// Mitsubishi GX Works2 project: BookEX6_5 Shift   PLC: Q06UDV

// global labels: Global
VAR_GLOBAL
  bVar0 AT M5000 : BOOL;
  abArray0 AT M5010 : ARRAY [0..49] OF BOOL;
  sStr0 AT D5000 : STRING[199];
  sStr1 AT D5100 : STRING[199];
  sStr2 AT D5200 : STRING[199];
  sStr3 AT D5300 : STRING[199];
  sStr4 AT D5400 : STRING[199];
  sStr5 AT D5500 : STRING[199];
  sStr6 AT D5600 : STRING[199];
  sStr7 AT D5700 : STRING[199];
  sStr8 AT D5800 : STRING[199];
  sStr9 AT D5900 : STRING[199];
  iVar0 AT D4500 : INT;
  iVar1 AT D4501 : INT;
  iVar2 AT D4502 : INT;
  iVar3 AT D4503 : INT;
  iVar4 AT D4504 : INT;
  iVar5 AT D4505 : INT;
  iVar6 AT D4506 : INT;
  iVar7 AT D4507 : INT;
  iVar8 AT D4508 : INT;
  iVar9 AT D4509 : INT;
  dVar0 AT D4510 : DINT;
  dVar1 AT D4512 : DINT;
  dVar2 AT D4514 : DINT;
  dVar3 AT D4516 : DINT;
  dVar4 AT D4518 : DINT;
  dVar5 AT D4520 : DINT;
  dVar6 AT D4522 : DINT;
  dVar7 AT D4524 : DINT;
  dVar8 AT D4526 : DINT;
  dVar9 AT D4528 : DINT;
  wVar0 AT D4530 : WORD;
  wVar1 AT D4531 : WORD;
  wVar2 AT D4532 : WORD;
  wVar3 AT D4533 : WORD;
  wVar4 AT D4534 : WORD;
  wVar5 AT D4535 : WORD;
  wVar6 AT D4536 : WORD;
  wVar7 AT D4537 : WORD;
  wVar8 AT D4538 : WORD;
  wVar9 AT D4539 : WORD;
  dwVar0 AT D4540 : DWORD;
  dwVar1 AT D4542 : DWORD;
  dwVar2 AT D4544 : DWORD;
  dwVar3 AT D4546 : DWORD;
  dwVar4 AT D4548 : DWORD;
  dwVar5 AT D4550 : DWORD;
  dwVar6 AT D4552 : DWORD;
  dwVar7 AT D4554 : DWORD;
  dwVar8 AT D4556 : DWORD;
  dwVar9 AT D4558 : DWORD;
  fsVar0 AT D4560 : REAL;
  fsVar1 AT D4562 : REAL;
  fsVar2 AT D4564 : REAL;
  fsVar3 AT D4566 : REAL;
  fsVar4 AT D4568 : REAL;
  fsVar5 AT D4570 : REAL;
  fsVar6 AT D4572 : REAL;
  fsVar7 AT D4574 : REAL;
  fsVar8 AT D4576 : REAL;
  fsVar9 AT D4578 : REAL;
  fdVar0 AT D4580 : LREAL;
  tTime0 AT D4620 : TIME;
  tTime1 AT D4622 : TIME;
  tTime2 AT D4624 : TIME;
  tTime3 AT D4626 : TIME;
  tTime4 AT D4628 : TIME;
  tTime5 AT D4630 : TIME;
  tTime6 AT D4632 : TIME;
  tTime7 AT D4634 : TIME;
  tTime8 AT D4636 : TIME;
  tTime9 AT D4638 : TIME;
  tTime10 AT D4640 : TIME;
  bVar1 AT M5001 : BOOL;
  bVar2 AT M5002 : BOOL;
  bVar3 AT M5003 : BOOL;
  bVar4 AT M5004 : BOOL;
  bVar5 AT M5005 : BOOL;
  bVar6 AT M5006 : BOOL;
  bVar7 AT M5007 : BOOL;
  bVar8 AT M5008 : BOOL;
  bVar9 AT M5009 : BOOL;
  abArray1 AT M5060 : ARRAY [0..49] OF BOOL;
  abArray2 AT M5110 : ARRAY [0..49] OF BOOL;
  abArray3 AT M5160 : ARRAY [0..49] OF BOOL;
  abArray4 AT M5210 : ARRAY [0..49] OF BOOL;
  abArray5 AT M5260 : ARRAY [0..49] OF BOOL;
  abArray6 AT M5310 : ARRAY [0..49] OF BOOL;
  abArray7 AT M5360 : ARRAY [0..49] OF BOOL;
  abArray8 AT M5410 : ARRAY [0..49] OF BOOL;
  abArray9 AT M5460 : ARRAY [0..49] OF BOOL;
  fdVar1 AT D4584 : LREAL;
  fdVar2 AT D4588 : LREAL;
  fdVar3 AT D4592 : LREAL;
  fdVar4 AT D4596 : LREAL;
  fdVar5 AT D4600 : LREAL;
  fdVar6 AT D4604 : LREAL;
  fdVar7 AT D4608 : LREAL;
  fdVar8 AT D4612 : LREAL;
  fdVar9 AT D4616 : LREAL;
  adwD10 AT D10 : ARRAY [0..9] OF DWORD;
  awD10 AT D10 : ARRAY [0..19] OF WORD;
  abM10 AT M10 : ARRAY [0..7] OF BOOL;
END_VAR
// user libraries (not included): HMI

PROGRAM ExMask
(* structured ladder/FBD written out as ST: instructions are called as NAME(EN, inputs, outputs); _pN, _eN, _tN stand for wires *)
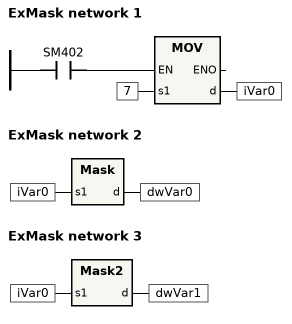
(* network 1 *)
MOV(SM402, 7, iVar0);
(* network 2 *)
dwVar0 := Mask(iVar0);
(* network 3 *)
dwVar1 := Mask2(iVar0);
END_PROGRAM

PROGRAM ExNewSHR_SHL
VAR
  ix : INT;
  iy : INT;
END_VAR
;

IF LDP(TRUE, SM412) THEN
	dwVar0 := H80000000; 
	dwVar1 := H80000000; 
	dwVar2 := H00000001; 
	dwVar3 := H00000001; 
	wVar0 := H8000;
	wVar1 := H0001;
	wVar2 := H8000;
	wVar3 := H0001;
	CASE ix OF
		0 :  (* 초기화 *)
				ix := 1;
		1..16 : (* Shift Bit *)
				dwVar0 := newDSHR(dwVar0, ix);
				abM10[0] := SM700;
				dwVar1 := newDSHR1(dwVar1, ix);
				abM10[1] := SM700;
				dwVar2 := newDSHL(dwVar2, ix);
				abM10[2] := SM700;
				dwVar3 := newDSHL1(dwVar3, ix);
				abM10[3] := SM700;
				wVar0 := newSHR(wVar0, ix);
				abM10[4] := SM700;
				wVar1 := newSHL(wVar1, ix);
				abM10[5] := SM700;
				wVar2 := newSHR1(wVar2, ix);
				abM10[6] := SM700;
				wVar3 := newSHL1(wVar3, ix);
				abM10[7] := SM700;
				ix := ix+1;
		17..32 : (* Shift Bit *)
				dwVar0 := newDSHR(dwVar0, ix);
				abM10[0] := SM700;
				dwVar1 := newDSHR1(dwVar1, ix);
				abM10[1] := SM700;
				dwVar2 := newDSHL(dwVar2, ix);
				abM10[2] := SM700;
				dwVar3 := newDSHL1(dwVar3, ix);
				abM10[3] := SM700;
				ix := ix+1;
		ELSE  
				ix := 0;
	END_CASE;
	adwD10[0] := dwVar0;
	adwD10[1] := dwVar1;
	adwD10[2] := dwVar2;
	adwD10[3] := dwVar3;
	awD10[8] := wVar0;
	awD10[9] := wVar1;
	awD10[10] := wVar2;
	awD10[11] := wVar3;
END_IF;
END_PROGRAM

PROGRAM ExROL
(* structured ladder/FBD written out as ST: instructions are called as NAME(EN, inputs, outputs); _pN, _eN, _tN stand for wires *)
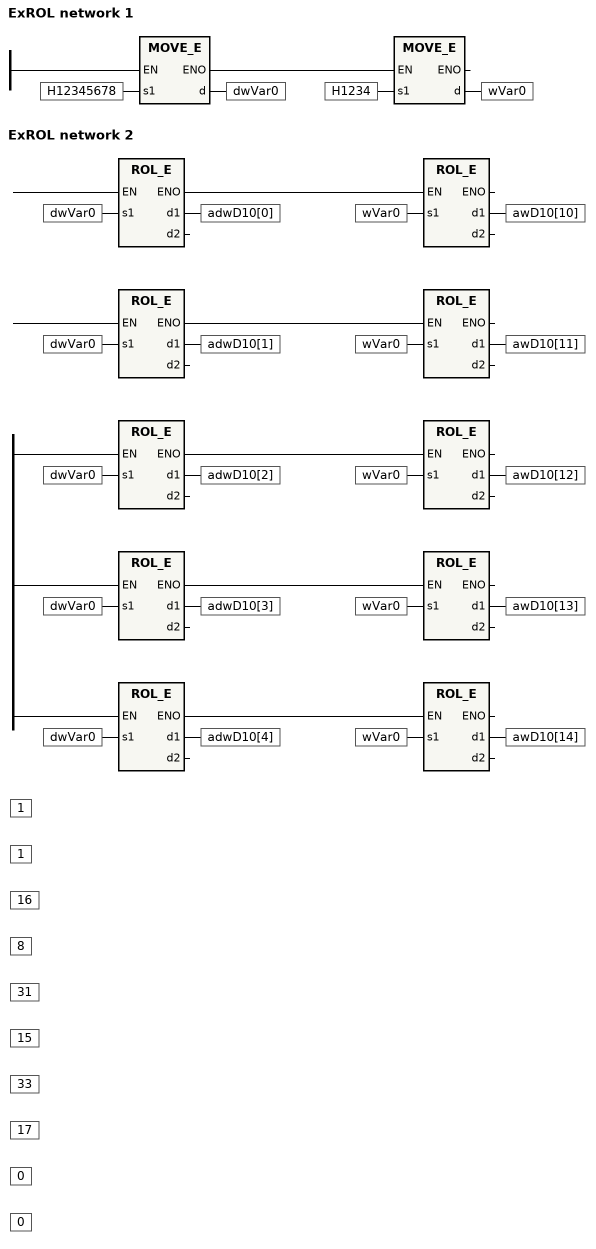
(* network 1 *)
_e1 := MOVE_E(TRUE, H12345678, dwVar0);
MOVE_E(_e1, H1234, wVar0);
(* network 2 *)
_e1 := ROL_E(TRUE, dwVar0, adwD10[0], _open);
ROL_E(_e1, wVar0, awD10[10], _open);
_e2 := ROL_E(TRUE, dwVar0, adwD10[1], _open);
ROL_E(_e2, wVar0, awD10[11], _open);
_e3 := ROL_E(TRUE, dwVar0, adwD10[2], _open);
ROL_E(_e3, wVar0, awD10[12], _open);
_e4 := ROL_E(TRUE, dwVar0, adwD10[3], _open);
ROL_E(_e4, wVar0, awD10[13], _open);
_e5 := ROL_E(TRUE, dwVar0, adwD10[4], _open);
ROL_E(_e5, wVar0, awD10[14], _open);
(* not connected to any output: 1, 1, 16, 8, 31, 15, 33, 17, 0, 0 *)
END_PROGRAM

PROGRAM ExROR
(* structured ladder/FBD written out as ST: instructions are called as NAME(EN, inputs, outputs); _pN, _eN, _tN stand for wires *)
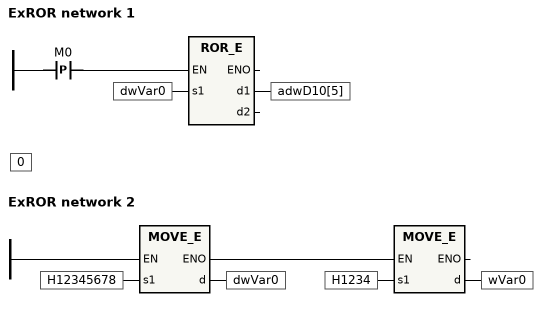
(* network 1 *)
ROR_E(LDP(TRUE, M0), dwVar0, adwD10[5], _open);
(* not connected to any output: 0 *)
(* network 2 *)
_e1 := MOVE_E(TRUE, H12345678, dwVar0);
MOVE_E(_e1, H1234, wVar0);
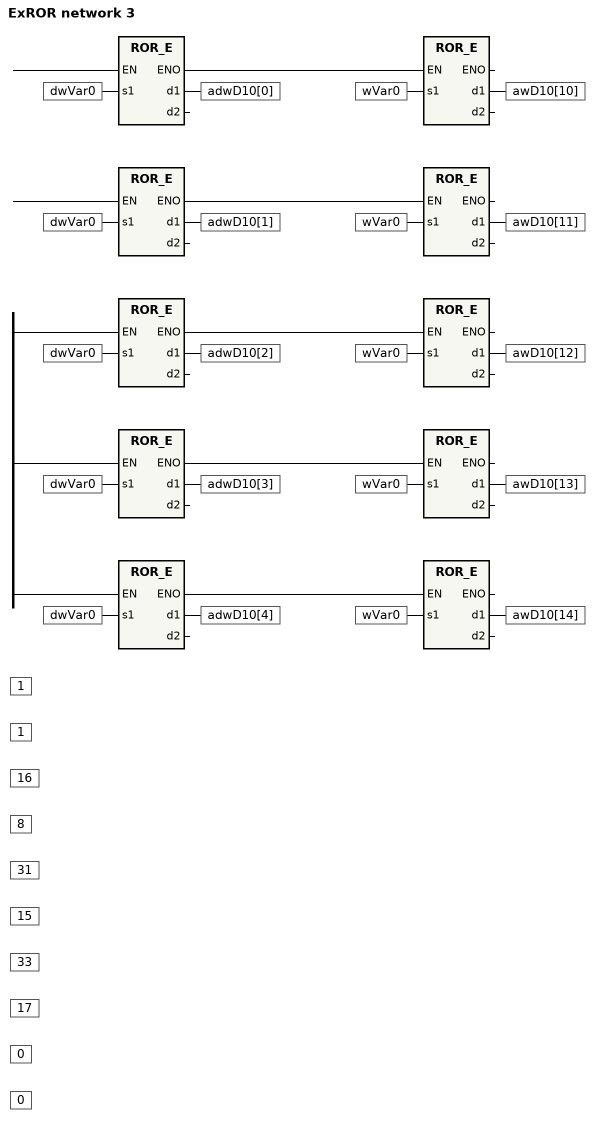
(* network 3 *)
_e1 := ROR_E(TRUE, dwVar0, adwD10[0], _open);
ROR_E(_e1, wVar0, awD10[10], _open);
_e2 := ROR_E(TRUE, dwVar0, adwD10[1], _open);
ROR_E(_e2, wVar0, awD10[11], _open);
_e3 := ROR_E(TRUE, dwVar0, adwD10[2], _open);
ROR_E(_e3, wVar0, awD10[12], _open);
_e4 := ROR_E(TRUE, dwVar0, adwD10[3], _open);
ROR_E(_e4, wVar0, awD10[13], _open);
_e5 := ROR_E(TRUE, dwVar0, adwD10[4], _open);
ROR_E(_e5, wVar0, awD10[14], _open);
(* not connected to any output: 1, 1, 16, 8, 31, 15, 33, 17, 0, 0 *)
END_PROGRAM

PROGRAM ExROR_ROL
VAR
  ix : INT;
  iy : INT;
END_VAR
;
IF LDP(TRUE, SM412) THEN
	dwVar0 := H80000000; 
	dwVar1 := H80000000; 
	dwVar2 := H00000001; 
	dwVar3 := H00000001; 
	wVar0 := H8000;
	wVar1 := H0001;
	wVar2 := H8000;
	wVar3 := H0001;
	CASE ix OF
		0 :  (* 초기화 *)
				ix := 1;
		1..16 : (* Shift Bit *)
				FOR iy := 1 TO ix DO  
					ROR_E(TRUE, dwVar0, 1, dwVar0);
				END_FOR;  
				abM10[0] := SM700;
				DROR(TRUE, ix, dwVar1);
				abM10[1] := SM700;
				FOR iy := 1 TO ix DO  
					ROL_E(TRUE, dwVar2, 1, dwVar2);
				END_FOR;  
				abM10[2] := SM700;
				DROL(TRUE, ix, dwVar3);  
				abM10[3] := SM700;
				FOR iy := 1 TO ix DO  
					ROR_E(TRUE, wVar0, 1, wVar0);
				END_FOR;  
				abM10[4] := SM700;
				FOR iy := 1 TO ix DO  
					ROL_E(TRUE, wVar1, 1, wVar1);
				END_FOR;  
				abM10[5] := SM700;
				ROR(TRUE, ix, wVar2);
				abM10[6] := SM700;
				ROL(TRUE, ix, wVar3);
				abM10[7] := SM700;
				ix := ix+1;
		17..32 : (* Shift Bit *)
				FOR iy := 1 TO ix DO  
					ROR_E(TRUE, dwVar0, 1, dwVar0);
				END_FOR;  
				abM10[0] := SM700;
				DROR(TRUE, ix, dwVar1);
				abM10[1] := SM700;
				FOR iy := 1 TO ix DO  
					ROL_E(TRUE, dwVar2, 1, dwVar2);
				END_FOR;  
				abM10[2] := SM700;
				DROL(TRUE, ix, dwVar3);  
				abM10[3] := SM700;
				ix := ix+1;
		ELSE  
				ix := 0;
	END_CASE;
	adwD10[0] := dwVar0;
	adwD10[1] := dwVar1;
	adwD10[2] := dwVar2;
	adwD10[3] := dwVar3;
	awD10[8] := wVar0;
	awD10[9] := wVar1;
	awD10[10] := wVar2;
	awD10[11] := wVar3;
END_IF;
END_PROGRAM

PROGRAM ExSHL
(* structured ladder/FBD written out as ST: instructions are called as NAME(EN, inputs, outputs); _pN, _eN, _tN stand for wires *)
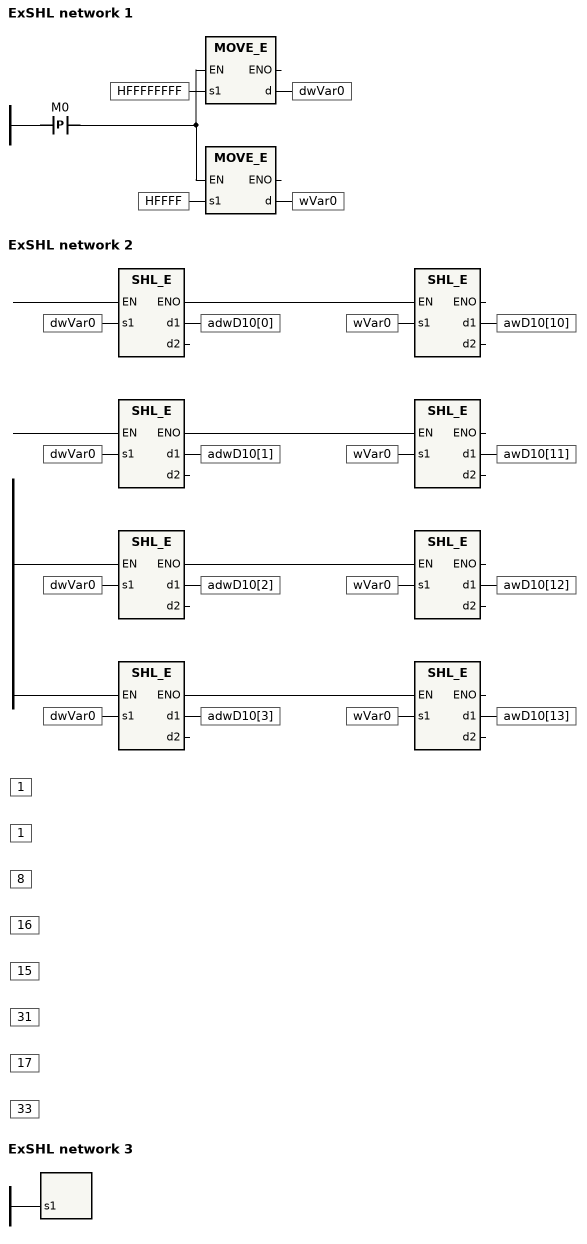
(* network 1 *)
_p1 := LDP(TRUE, M0);
MOVE_E(_p1, HFFFFFFFF, dwVar0);
MOVE_E(_p1, HFFFF, wVar0);
(* network 2 *)
_e1 := SHL_E(TRUE, dwVar0, adwD10[0], _open);
SHL_E(_e1, wVar0, awD10[10], _open);
_e2 := SHL_E(TRUE, dwVar0, adwD10[1], _open);
SHL_E(_e2, wVar0, awD10[11], _open);
_e3 := SHL_E(TRUE, dwVar0, adwD10[2], _open);
SHL_E(_e3, wVar0, awD10[12], _open);
_e4 := SHL_E(TRUE, dwVar0, adwD10[3], _open);
SHL_E(_e4, wVar0, awD10[13], _open);
(* not connected to any output: 1, 1, 8, 16, 15, 31, 17, 33 *)
(* network 3 *)
(* element kind 10  <- TRUE *)
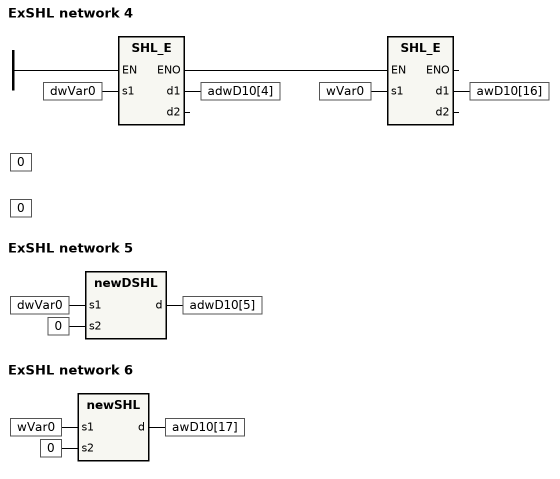
(* network 4 *)
_e1 := SHL_E(TRUE, dwVar0, adwD10[4], _open);
SHL_E(_e1, wVar0, awD10[16], _open);
(* not connected to any output: 0, 0 *)
(* network 5 *)
adwD10[5] := newDSHL(dwVar0, 0);
(* network 6 *)
awD10[17] := newSHL(wVar0, 0);
END_PROGRAM

PROGRAM ExSHR
(* structured ladder/FBD written out as ST: instructions are called as NAME(EN, inputs, outputs); _pN, _eN, _tN stand for wires *)
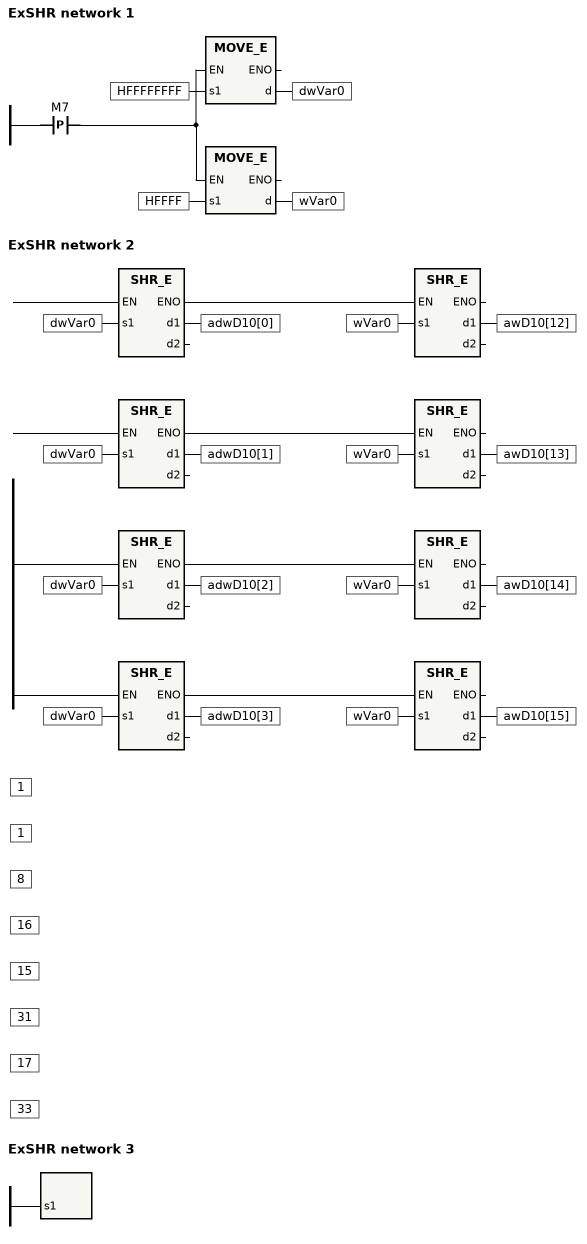
(* network 1 *)
_p1 := LDP(TRUE, M7);
MOVE_E(_p1, HFFFFFFFF, dwVar0);
MOVE_E(_p1, HFFFF, wVar0);
(* network 2 *)
_e1 := SHR_E(TRUE, dwVar0, adwD10[0], _open);
SHR_E(_e1, wVar0, awD10[12], _open);
_e2 := SHR_E(TRUE, dwVar0, adwD10[1], _open);
SHR_E(_e2, wVar0, awD10[13], _open);
_e3 := SHR_E(TRUE, dwVar0, adwD10[2], _open);
SHR_E(_e3, wVar0, awD10[14], _open);
_e4 := SHR_E(TRUE, dwVar0, adwD10[3], _open);
SHR_E(_e4, wVar0, awD10[15], _open);
(* not connected to any output: 1, 1, 8, 16, 15, 31, 17, 33 *)
(* network 3 *)
(* element kind 10  <- TRUE *)
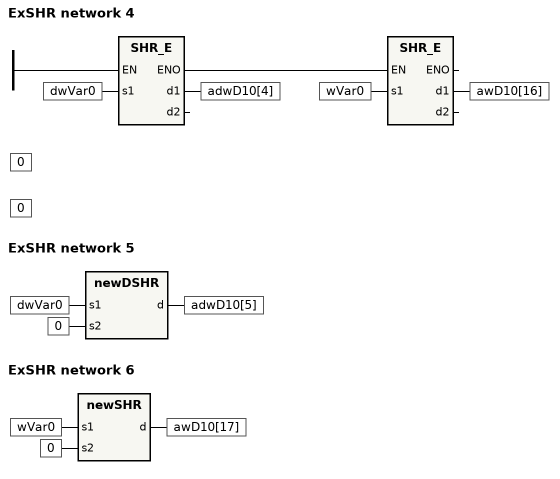
(* network 4 *)
_e1 := SHR_E(TRUE, dwVar0, adwD10[4], _open);
SHR_E(_e1, wVar0, awD10[16], _open);
(* not connected to any output: 0, 0 *)
(* network 5 *)
adwD10[5] := newDSHR(dwVar0, 0);
(* network 6 *)
awD10[17] := newSHR(wVar0, 0);
END_PROGRAM

PROGRAM ExSHR_SHL
VAR
  ix : INT;
  iy : INT;
END_VAR
;

IF LDP(TRUE, SM412) THEN
	dwVar0 := H80000000;
	dwVar1 := H00000001;
	wVar0 := H8000;
	wVar1 := H0001;
	CASE ix OF
		0 :  (* 초기화 *)
				ix := 1;
		1..16 : (* Shift Bit *)
				FOR iy := 1 TO ix DO  
					dwVar0 := SHR(dwVar0, 1);
				END_FOR;  
				abM10[0] := SM700;
				FOR iy := 1 TO ix DO 
					dwVar1 := SHL(dwVar1, 1);
				END_FOR;
				abM10[1] := SM700;
				FOR iy := 1 TO ix DO 
					wVar0 := SHR(wVar0, 1);
				END_FOR;
				abM10[2] := SM700;
				FOR iy := 1 TO ix DO 
					wVar1 := SHL(wVar1, 1);
				END_FOR;
				abM10[3] := SM700;
				ix := ix+1;
		17..32 : (* Shift Bit *)
				FOR iy := 1 TO ix DO  
					dwVar0 := SHR(dwVar0, 1);
				END_FOR;  
				abM10[0] := SM700;
				FOR iy := 1 TO ix DO 
					dwVar1 := SHL(dwVar1, 1);
				END_FOR;
				abM10[1] := SM700;
				ix := ix+1;
		ELSE  
				ix := 0;
	END_CASE;
	adwD10[0] := dwVar0;
	adwD10[1] := dwVar1;
	awD10[6] := wVar0;
	awD10[7] := wVar1;
END_IF;
END_PROGRAM

PROGRAM ExTemp
VAR
  Mov4WORD_1 : Mov4WORD;
  Mov4DWORD_1 : Mov4DWORD;
END_VAR
(* structured ladder/FBD written out as ST: instructions are called as NAME(EN, inputs, outputs); _pN, _eN, _tN stand for wires *)
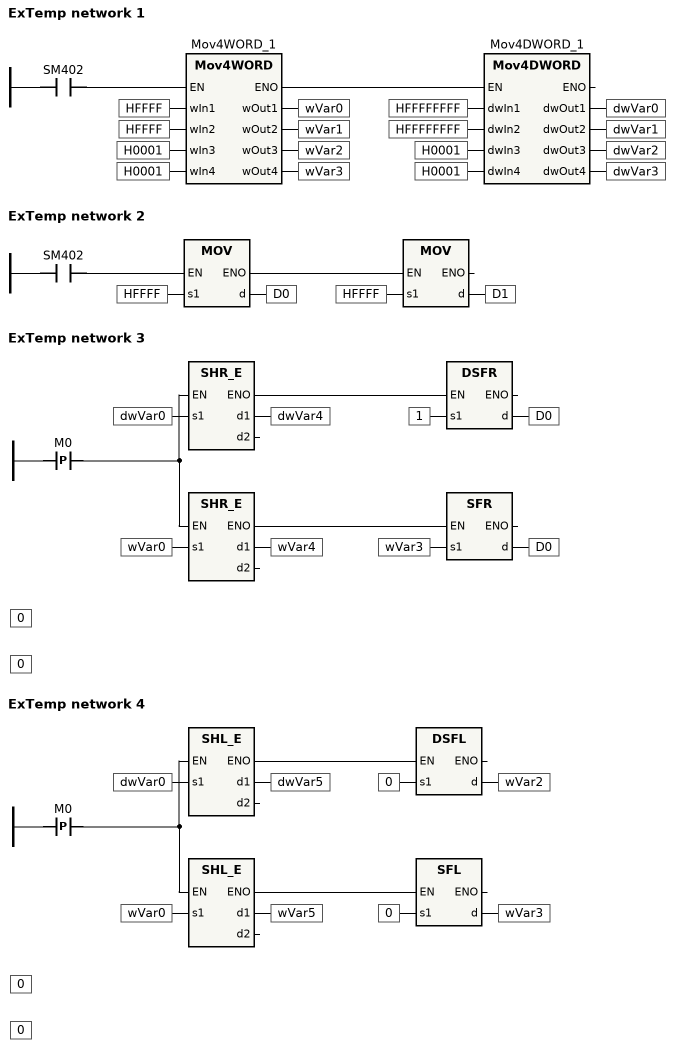
(* network 1 *)
Mov4WORD_1(EN := SM402, wIn1 := HFFFF, wIn2 := HFFFF, wIn3 := H0001, wIn4 := H0001, wOut1 => wVar0, wOut2 => wVar1, wOut3 => wVar2, wOut4 => wVar3);
Mov4DWORD_1(EN := Mov4WORD_1.ENO, dwIn1 := HFFFFFFFF, dwIn2 := HFFFFFFFF, dwIn3 := H0001, dwIn4 := H0001, dwOut1 => dwVar0, dwOut2 => dwVar1, dwOut3 => dwVar2, dwOut4 => dwVar3);
(* network 2 *)
_e1 := MOV(SM402, HFFFF, D0);
MOV(_e1, HFFFF, D1);
(* network 3 *)
_p1 := LDP(TRUE, M0);
_e2 := SHR_E(_p1, dwVar0, dwVar4, _open);
DSFR(_e2, 1, D0);
_e3 := SHR_E(_p1, wVar0, wVar4, _open);
SFR(_e3, wVar3, D0);
(* not connected to any output: 0, 0 *)
(* network 4 *)
_p1 := LDP(TRUE, M0);
_e2 := SHL_E(_p1, dwVar0, dwVar5, _open);
DSFL(_e2, 0, wVar2);
_e3 := SHL_E(_p1, wVar0, wVar5, _open);
SFL(_e3, 0, wVar3);
(* not connected to any output: 0, 0 *)
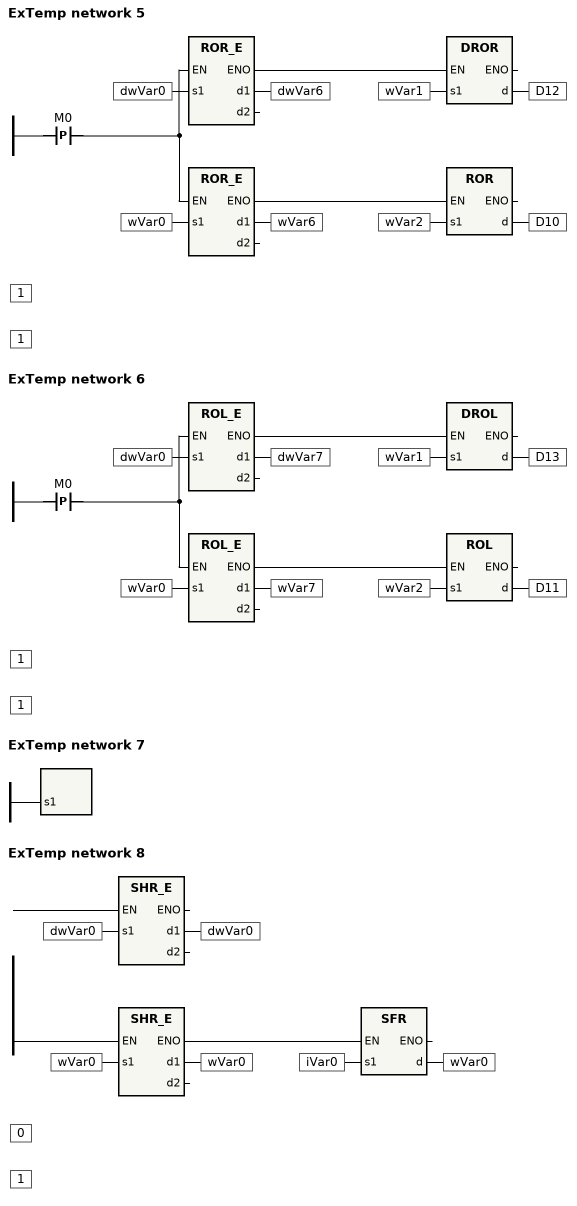
(* network 5 *)
_p1 := LDP(TRUE, M0);
_e2 := ROR_E(_p1, dwVar0, dwVar6, _open);
DROR(_e2, wVar1, D12);
_e3 := ROR_E(_p1, wVar0, wVar6, _open);
ROR(_e3, wVar2, D10);
(* not connected to any output: 1, 1 *)
(* network 6 *)
_p1 := LDP(TRUE, M0);
_e2 := ROL_E(_p1, dwVar0, dwVar7, _open);
DROL(_e2, wVar1, D13);
_e3 := ROL_E(_p1, wVar0, wVar7, _open);
ROL(_e3, wVar2, D11);
(* not connected to any output: 1, 1 *)
(* network 7 *)
(* element kind 10  <- TRUE *)
(* network 8 *)
SHR_E(TRUE, dwVar0, dwVar0, _open);
_e1 := SHR_E(TRUE, wVar0, wVar0, _open);
SFR(_e1, iVar0, wVar0);
(* not connected to any output: 0, 1 *)
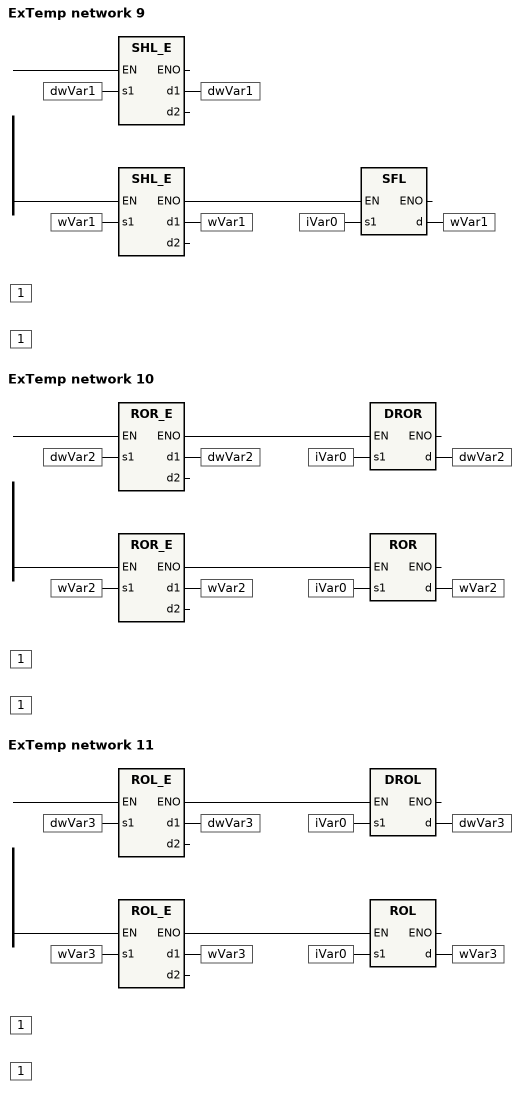
(* network 9 *)
SHL_E(TRUE, dwVar1, dwVar1, _open);
_e1 := SHL_E(TRUE, wVar1, wVar1, _open);
SFL(_e1, iVar0, wVar1);
(* not connected to any output: 1, 1 *)
(* network 10 *)
_e1 := ROR_E(TRUE, dwVar2, dwVar2, _open);
DROR(_e1, iVar0, dwVar2);
_e2 := ROR_E(TRUE, wVar2, wVar2, _open);
ROR(_e2, iVar0, wVar2);
(* not connected to any output: 1, 1 *)
(* network 11 *)
_e1 := ROL_E(TRUE, dwVar3, dwVar3, _open);
DROL(_e1, iVar0, dwVar3);
_e2 := ROL_E(TRUE, wVar3, wVar3, _open);
ROL(_e2, iVar0, wVar3);
(* not connected to any output: 1, 1 *)
END_PROGRAM

PROGRAM extest
VAR
  ix : INT;
  iy : INT;
  Temp0 : DWORD;
  Temp1 : DWORD;
  wTemp0 : WORD;
  wTemp1 : WORD;
END_VAR
;

IF LDP(TRUE, M9) THEN
	dwVar0 := H80000000; 
	dwVar1 := H00000001; 
	wVar0 := H8000;
	wVar1 := H0001;
	wVar2 := H8000;
	wVar3 := H0001;
	CASE ix OF
		0 :  (* 초기화 *)
				ix := 1;
		1..16 : (* Shift Bit *)
				dwVar0 := newDSHR(dwVar0, ix);
				abM10[0] := SM700;
				dwVar1 := newDSHL(dwVar1, ix);
				abM10[1] := SM700;
				Temp0 := Mask(32-ix);
				Temp1 := Mask(ix);
 			 	wVar0 := newSHR(wVar0, ix);
				abM10[2] := SM700;
				wVar1 := newSHL(wVar1, ix);
				abM10[3] := SM700;
				wVar2 := newSHR1(wVar2, ix);
				abM10[4] := SM700;
				wVar3 := newSHL1(wVar3, ix);
				abM10[5] := SM700; 
				wTemp0 := DWORD_TO_WORD(Mask(16-ix));
				wTemp1 := DWORD_TO_WORD(Mask(ix));
				ix := ix+1;
		17..32 : (* Shift Bit *)
				dwVar0 := newDSHR(dwVar0, ix);
				abM10[0] := SM700;
				dwVar1 := newDSHL(dwVar1, ix);
				abM10[1] := SM700;
				Temp0 := Mask(32-ix);
				Temp1 := Mask(ix);
				ix := ix+1;
		ELSE  
				ix := 0;
	END_CASE;
	adwD10[0] := dwVar0;
	adwD10[1] := dwVar1;
	adwD10[2] := Temp0 ;
	adwD10[3] := Temp1 ;
	awD10[12] := wTemp0 ;
	awD10[13] := wTemp1 ;
    awD10[8] := wVar0;
	awD10[9] := wVar1;
	awD10[10] := wVar2;
	awD10[11] := wVar3; 
END_IF;
END_PROGRAM

PROGRAM ExWireTXD
VAR
  Mov4WORD_1 : Mov4WORD;
  wireTXD_1 : wireTXD;
  HMI02_1 : HMI02;
END_VAR
(* structured ladder/FBD written out as ST: instructions are called as NAME(EN, inputs, outputs); _pN, _eN, _tN stand for wires *)
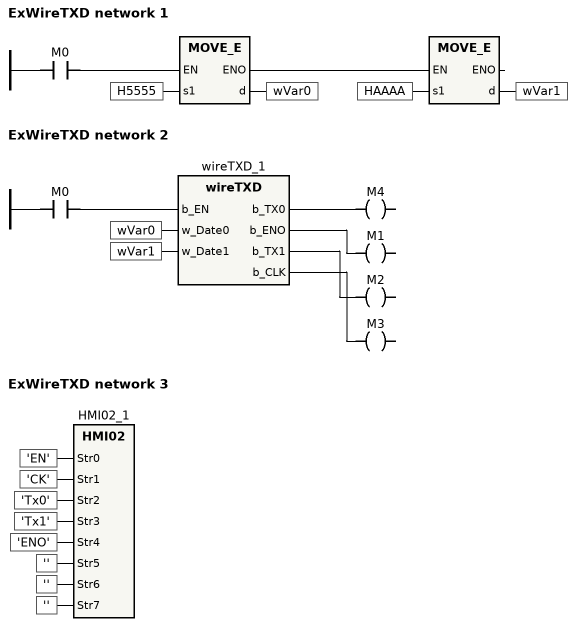
(* network 1 *)
_e1 := MOVE_E(M0, H5555, wVar0);
MOVE_E(_e1, HAAAA, wVar1);
(* network 2 *)
wireTXD_1(b_EN := M0, w_Date0 := wVar0, w_Date1 := wVar1);
M4 := wireTXD_1.b_TX0;
M1 := wireTXD_1.b_ENO;
M2 := wireTXD_1.b_TX1;
M3 := wireTXD_1.b_CLK;
(* network 3 *)
HMI02_1(Str0 := 'EN', Str1 := 'CK', Str2 := 'Tx0', Str3 := 'Tx1', Str4 := 'ENO', Str5 := '', Str6 := '', Str7 := '');
END_PROGRAM

FUNCTION Mask
VAR
  Temp : DWORD;
END_VAR
VAR_INPUT
  i_N : INT;
END_VAR
;
CASE i_N OF
	0 : Temp := 0;
	1 : Temp := H00000001;
	2 : Temp := H00000003;
	3 : Temp := H00000007;
	4 : Temp := H0000000F;
	5 : Temp := H0000001F;
	6 : Temp := H0000003F;
	7 : Temp := H0000007F;
	8 : Temp := H000000FF;
	9 : Temp := H000001FF;
	10 : Temp := H000003FF;
	11 : Temp := H000007FF;
	12 : Temp := H00000FFF;
	13 : Temp := H00001FFF;
	14 : Temp := H00003FFF;
	15 : Temp := H00007FFF;
	16 : Temp := H0000FFFF;
	17 : Temp := H0001FFFF;
	18 : Temp := H0003FFFF;
	19 : Temp := H0007FFFF;
	20 : Temp := H000FFFFF;
	21 : Temp := H001FFFFF;
	22 : Temp := H003FFFFF;
	23 : Temp := H007FFFFF;
	24 : Temp := H00FFFFFF;
	25 : Temp := H01FFFFFF;
	26 : Temp := H03FFFFFF;
	27 : Temp := H07FFFFFF;
	28 : Temp := H0FFFFFFF;
	29 : Temp := H1FFFFFFF;
	30 : Temp := H3FFFFFFF;
	31 : Temp := H7FFFFFFF;
	32 : Temp := HFFFFFFFF;
END_CASE;

Mask := Temp;
END_FUNCTION

FUNCTION Mask2
VAR
  Temp : DWORD;
END_VAR
VAR_INPUT
  i_N : INT;
END_VAR
VAR
  ix : INT;
END_VAR
;
Temp := HFFFFFFFF;
FOR ix := 0 TO 31 - i_N DO
	Temp := SHR(Temp, 1);
END_FOR;
Mask2 := Temp;
END_FUNCTION

FUNCTION newDSHL
VAR_INPUT
  i_Cnt : INT;
  dw_Data : DWORD;
END_VAR
VAR
  Cnt : INT;
  Temp : DWORD;
  Org : DWORD;
END_VAR
;
Cnt := ABS(i_Cnt) MOD 32;
Org := dw_Data;
Temp := Mask(Cnt);
DROL(TRUE, Cnt, Org);
newDSHL :=  Org AND NOT Temp;
END_FUNCTION

FUNCTION newDSHL1
VAR_INPUT
  i_Cnt : INT;
  dw_Data : DWORD;
END_VAR
VAR
  Cnt : INT;
  Temp : DWORD;
  Org : DWORD;
END_VAR
;
Cnt := ABS(i_Cnt) MOD 32;
Org := dw_Data;
Temp := Mask(Cnt);
DROL(TRUE, Cnt, Org);
newDSHL1 :=  Org OR Temp;
END_FUNCTION

FUNCTION newDSHR
VAR_INPUT
  i_Cnt : INT;
  dw_Data : DWORD;
END_VAR
VAR
  Cnt : INT;
  Temp : DWORD;
  Org : DWORD;
END_VAR
;
Cnt := ABS(i_Cnt) MOD 32;
Org := dw_Data;
Temp := Mask(32-Cnt);
DROR(TRUE, Cnt, Org);
newDSHR :=  Org AND Temp;
END_FUNCTION

FUNCTION newDSHR1
VAR_INPUT
  i_Cnt : INT;
  dw_Data : DWORD;
END_VAR
VAR
  Cnt : INT;
  Temp : DWORD;
  Org : DWORD;
END_VAR
;
Cnt := ABS(i_Cnt) MOD 32;
Org := dw_Data;
Temp := Mask(32-Cnt);
DROR(TRUE, Cnt, Org);
newDSHR1 :=  Org OR NOT Temp;
END_FUNCTION

FUNCTION newSHL
VAR_INPUT
  i_Cnt : INT;
  w_Data : WORD;
END_VAR
VAR
  Cnt : INT;
  Temp : WORD;
  Org : WORD;
END_VAR
;
Cnt := ABS(i_Cnt) MOD 16;
Org := w_Data;
Temp := DWORD_TO_WORD(Mask(Cnt));
ROL(TRUE, Cnt, Org);
newSHL :=  Org AND NOT Temp;
END_FUNCTION

FUNCTION newSHL1
VAR_INPUT
  i_Cnt : INT;
  w_Data : WORD;
END_VAR
VAR
  Cnt : INT;
  Temp : WORD;
  Org : WORD;
  tVar1 : TIME;
  tVar2 : TIME;
  tVar3 : TIME;
  tVar4 : TIME;
  tVar5 : TIME;
  tVar6 : TIME;
  tVar7 : TIME;
  tVar8 : TIME;
  tVar9 : TIME;
  fVar0 : REAL;
  ddVar0 : DINT;
  iTemp : INT;
END_VAR
;
Cnt := ABS(i_Cnt) MOD 16;
Org := w_Data;
Temp := DWORD_TO_WORD(Mask(Cnt));
ROL(TRUE, Cnt, Org);
newSHL1 :=  Org OR Temp;
END_FUNCTION

FUNCTION newSHR
VAR_INPUT
  i_Cnt : INT;
  w_Data : WORD;
END_VAR
VAR
  Cnt : INT;
  Temp : WORD;
  Org : WORD;
END_VAR
;
Cnt := ABS(i_Cnt) MOD 16;
Org := w_Data;
Temp := DWORD_TO_WORD(Mask(16-Cnt));
ROR(TRUE, Cnt, Org);
newSHR :=  Org AND Temp;
END_FUNCTION

FUNCTION newSHR1
VAR_INPUT
  i_Cnt : INT;
  w_Data : WORD;
END_VAR
VAR
  Cnt : INT;
  Temp : WORD;
  Org : WORD;
END_VAR
;
Cnt := ABS(i_Cnt) MOD 16;
Org := w_Data;
Temp := DWORD_TO_WORD(Mask(16-Cnt));
ROR(TRUE, Cnt, Org);
newSHR1 :=  Org OR NOT Temp;
END_FUNCTION

FUNCTION_BLOCK wireTXD
VAR_INPUT
  b_EN : BOOL;
  w_Date0 : WORD;
END_VAR
VAR_OUTPUT
  b_TX0 : BOOL;
  b_ENO : BOOL;
END_VAR
VAR
  Phase : INT;
  wMaskBit : WORD;
  wTD1 : WORD;
  wTD0 : WORD;
END_VAR
VAR_INPUT
  w_Date1 : WORD;
END_VAR
VAR_OUTPUT
  b_TX1 : BOOL;
  b_CLK : BOOL;
END_VAR
;
IF NOT b_EN AND Phase = 0 THEN
	b_ENO := FALSE;
	b_CLK := TRUE;
	b_TX0 := TRUE;
	b_TX1 := TRUE;
	Phase := 0;
	RETURN;
END_IF;

b_ENO := TRUE;
CASE Phase OF
	0 :   
			b_CLK := TRUE;
			b_TX0 := TRUE;
			b_TX1 := TRUE;
			wTD0 := w_Date0;
			wTD1 := w_Date1;
			Phase := 1;
	1 : 
			b_CLK := FALSE;
			b_TX0 := TRUE;
			b_TX1 := TRUE;
			wMaskBit := H8000;
			Phase := 2;
	2..33 :  		
			b_TX0 := (wMaskBit AND wTD0) <> 0;
			b_TX1 := (wMaskBit AND wTD1) <> 0;
			IF (Phase MOD 2) = 0 THEN
    			b_CLK := TRUE;		
			ELSE 
	  			b_CLK := FALSE;		 
    			wMaskBit := SHR(wMaskBit, 1);
			END_IF;
			Phase := Phase + 1;
	34,36 :
			b_CLK := TRUE;
			b_TX0 := TRUE;
			b_TX1 := TRUE;
			Phase := Phase + 1;
	35,37 :
			b_CLK := FALSE;
			b_TX0 := TRUE;
			b_TX1 := TRUE;
			Phase := Phase + 1;
	ELSE  
			b_CLK := TRUE;
			b_TX0 := TRUE;
			b_TX1 := TRUE;
			Phase := 0;
END_CASE;
END_FUNCTION_BLOCK

PROGRAM ExTestSHR
VAR
  dwInitVar : DWORD;
  dwRes0 : DWORD;
  dwRes1 : DWORD;
  dwRes2 : DWORD;
  dwRes3 : DWORD;
  dwRes4 : DWORD;
  dwRes5 : DWORD;
  dwRes6 : DWORD;
  dwRes7 : DWORD;
  dwRes8 : DWORD;
  dwRes9 : DWORD;
  dwRes10 : DWORD;
  dwRes11 : DWORD;
  dwRes12 : DWORD;
  dwRes13 : DWORD;
  dwRes14 : DWORD;
  dwRes15 : DWORD;
  dwRes16 : DWORD;
  dwRes17 : DWORD;
  dwRes18 : DWORD;
  dwRes19 : DWORD;
  dwRes20 : DWORD;
  dwRes21 : DWORD;
  dwRes22 : DWORD;
  dwRes23 : DWORD;
  dwRes24 : DWORD;
  dwRes25 : DWORD;
  dwRes26 : DWORD;
  dwRes27 : DWORD;
  dwRes28 : DWORD;
  dwRes29 : DWORD;
  dwRes30 : DWORD;
  dwRes31 : DWORD;
  wInitVar : WORD;
  wRes0 : WORD;
  wRes1 : WORD;
  wRes2 : WORD;
  wRes3 : WORD;
  wRes4 : WORD;
  wRes5 : WORD;
  wRes6 : WORD;
  wRes7 : WORD;
  wRes8 : WORD;
  wRes9 : WORD;
  wRes10 : WORD;
  wRes11 : WORD;
  wRes12 : WORD;
  wRes13 : WORD;
  wRes14 : WORD;
  wRes15 : WORD;
  wRes16 : WORD;
  dwRes32 : DWORD;
  dwRes33 : DWORD;
  dwRes34 : DWORD;
  wRes17 : WORD;
  wRes18 : WORD;
  wRes19 : WORD;
  wRes20 : WORD;
  dwRes35 : DWORD;
  dwRes36 : DWORD;
  dwRes100 : DWORD;
  dwRes101 : DWORD;
  dwRes102 : DWORD;
  dwRes103 : DWORD;
  dwRes132 : DWORD;
  dwRes133 : DWORD;
  dwRes134 : DWORD;
  dwRes135 : DWORD;
  dwRes200 : DWORD;
  dwRes201 : DWORD;
  dwRes202 : DWORD;
  dwRes203 : DWORD;
  dwRes232 : DWORD;
  dwRes233 : DWORD;
  dwRes234 : DWORD;
  dwRes235 : DWORD;
  dwInitVar2 : DWORD;
  wInitVar2 : WORD;
END_VAR
(* structured ladder/FBD written out as ST: instructions are called as NAME(EN, inputs, outputs); _pN, _eN, _tN stand for wires *)
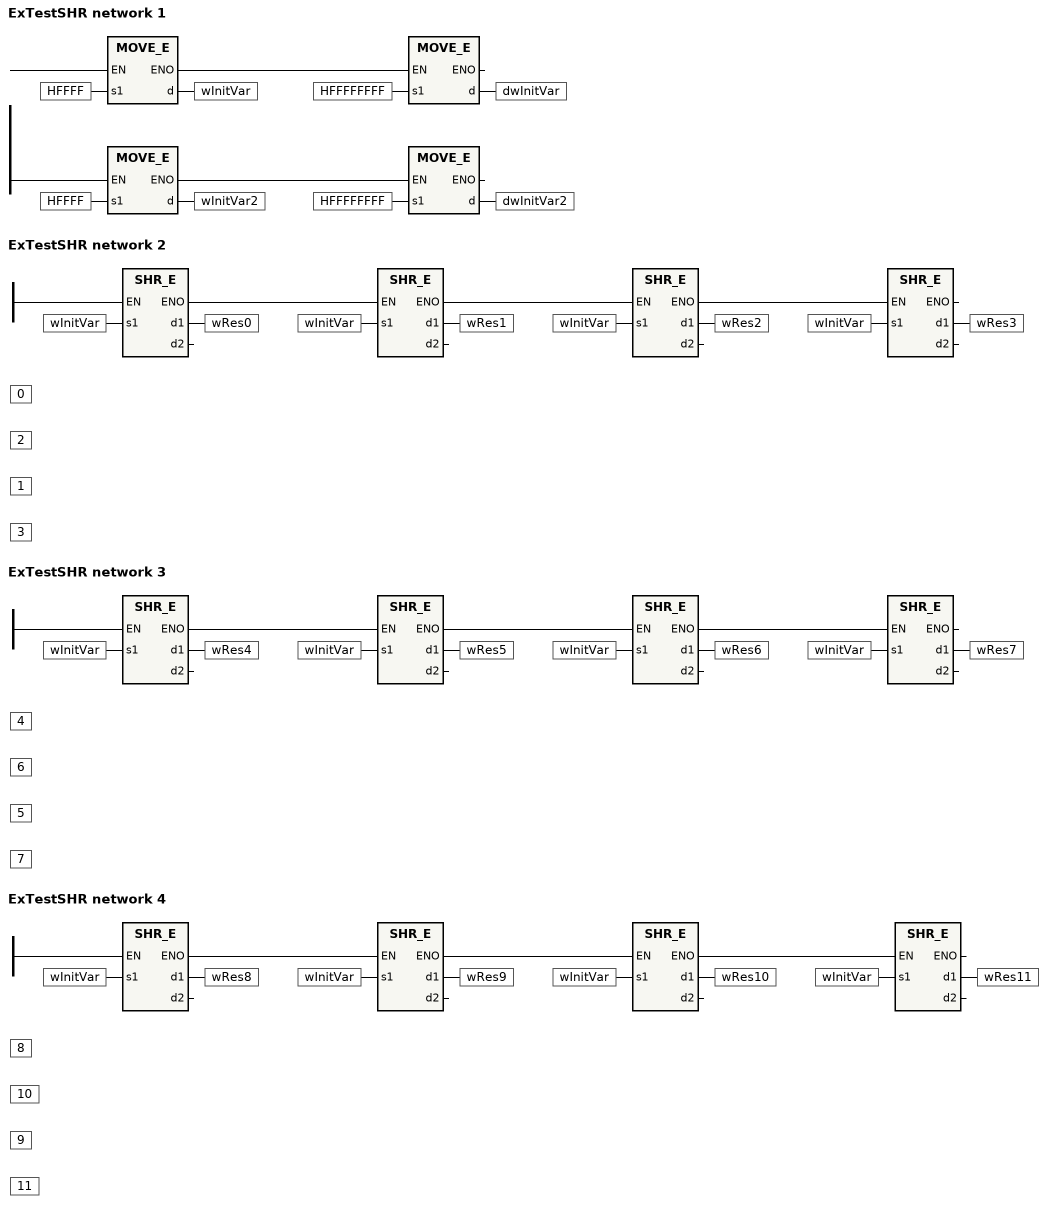
(* network 1 *)
_e1 := MOVE_E(TRUE, HFFFF, wInitVar);
MOVE_E(_e1, HFFFFFFFF, dwInitVar);
_e2 := MOVE_E(TRUE, HFFFF, wInitVar2);
MOVE_E(_e2, HFFFFFFFF, dwInitVar2);
(* network 2 *)
_e1 := SHR_E(TRUE, wInitVar, wRes0, _open);
_e2 := SHR_E(_e1, wInitVar, wRes1, _open);
_e3 := SHR_E(_e2, wInitVar, wRes2, _open);
SHR_E(_e3, wInitVar, wRes3, _open);
(* not connected to any output: 0, 2, 1, 3 *)
(* network 3 *)
_e1 := SHR_E(TRUE, wInitVar, wRes4, _open);
_e2 := SHR_E(_e1, wInitVar, wRes5, _open);
_e3 := SHR_E(_e2, wInitVar, wRes6, _open);
SHR_E(_e3, wInitVar, wRes7, _open);
(* not connected to any output: 4, 6, 5, 7 *)
(* network 4 *)
_e1 := SHR_E(TRUE, wInitVar, wRes8, _open);
_e2 := SHR_E(_e1, wInitVar, wRes9, _open);
_e3 := SHR_E(_e2, wInitVar, wRes10, _open);
SHR_E(_e3, wInitVar, wRes11, _open);
(* not connected to any output: 8, 10, 9, 11 *)
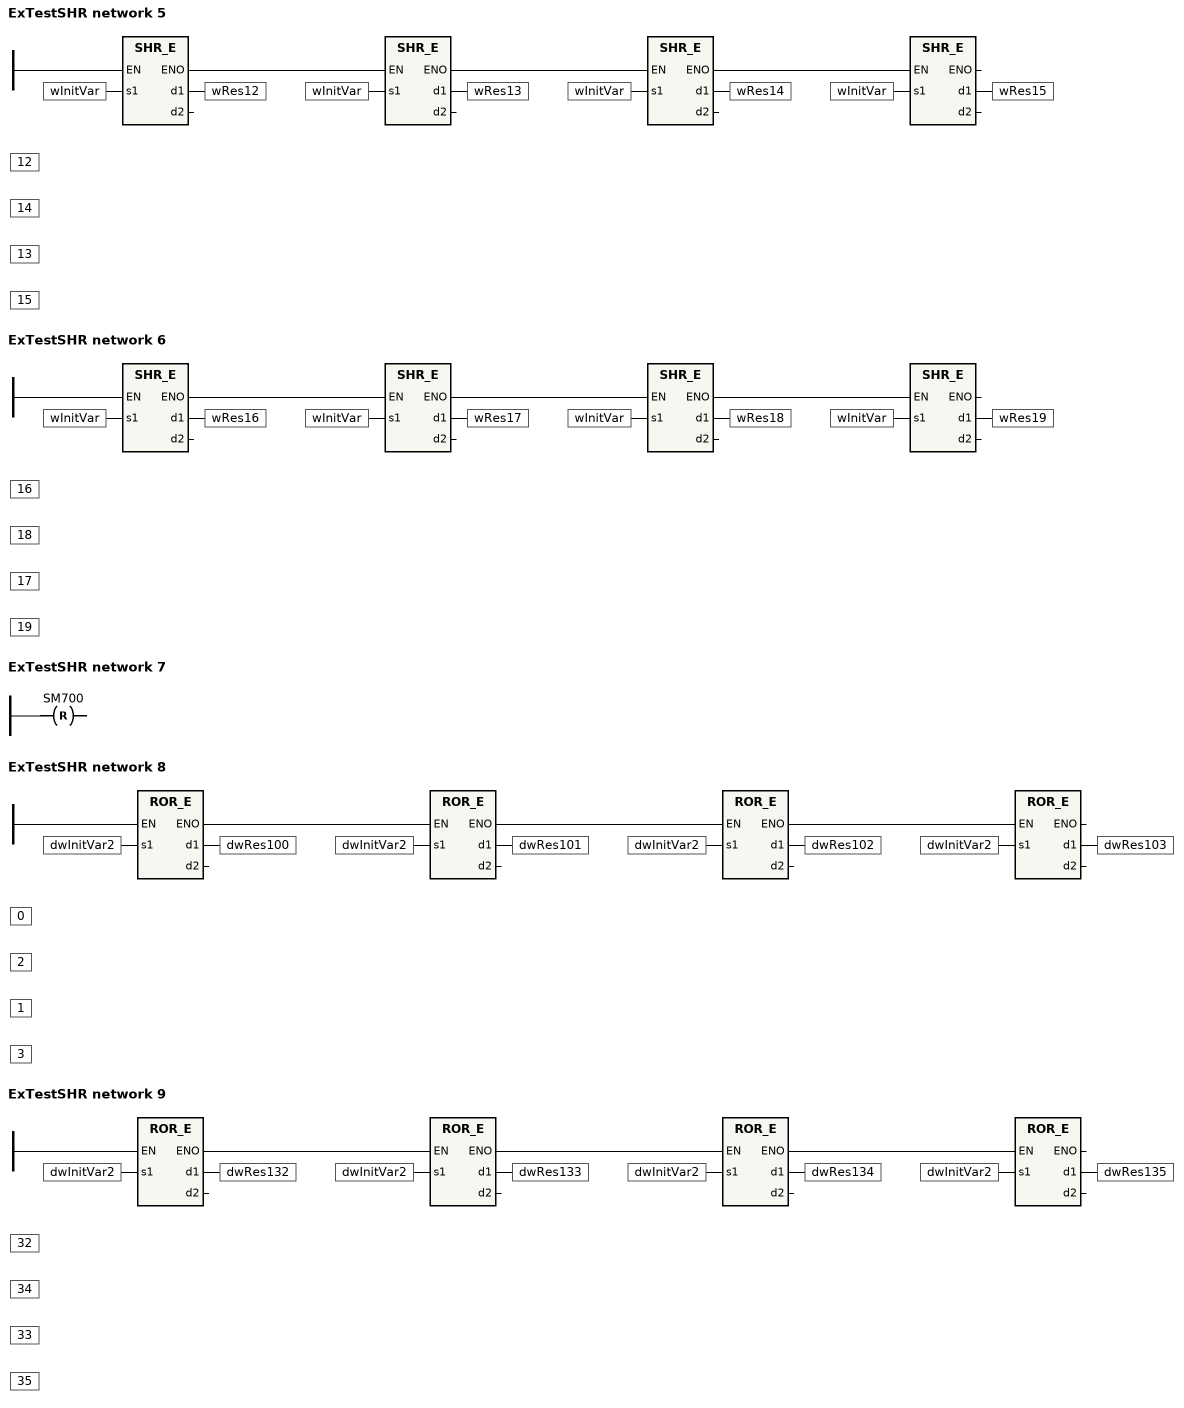
(* network 5 *)
_e1 := SHR_E(TRUE, wInitVar, wRes12, _open);
_e2 := SHR_E(_e1, wInitVar, wRes13, _open);
_e3 := SHR_E(_e2, wInitVar, wRes14, _open);
SHR_E(_e3, wInitVar, wRes15, _open);
(* not connected to any output: 12, 14, 13, 15 *)
(* network 6 *)
_e1 := SHR_E(TRUE, wInitVar, wRes16, _open);
_e2 := SHR_E(_e1, wInitVar, wRes17, _open);
_e3 := SHR_E(_e2, wInitVar, wRes18, _open);
SHR_E(_e3, wInitVar, wRes19, _open);
(* not connected to any output: 16, 18, 17, 19 *)
(* network 7 *)
RST(TRUE, SM700);
(* network 8 *)
_e1 := ROR_E(TRUE, dwInitVar2, dwRes100, _open);
_e2 := ROR_E(_e1, dwInitVar2, dwRes101, _open);
_e3 := ROR_E(_e2, dwInitVar2, dwRes102, _open);
ROR_E(_e3, dwInitVar2, dwRes103, _open);
(* not connected to any output: 0, 2, 1, 3 *)
(* network 9 *)
_e1 := ROR_E(TRUE, dwInitVar2, dwRes132, _open);
_e2 := ROR_E(_e1, dwInitVar2, dwRes133, _open);
_e3 := ROR_E(_e2, dwInitVar2, dwRes134, _open);
ROR_E(_e3, dwInitVar2, dwRes135, _open);
(* not connected to any output: 32, 34, 33, 35 *)
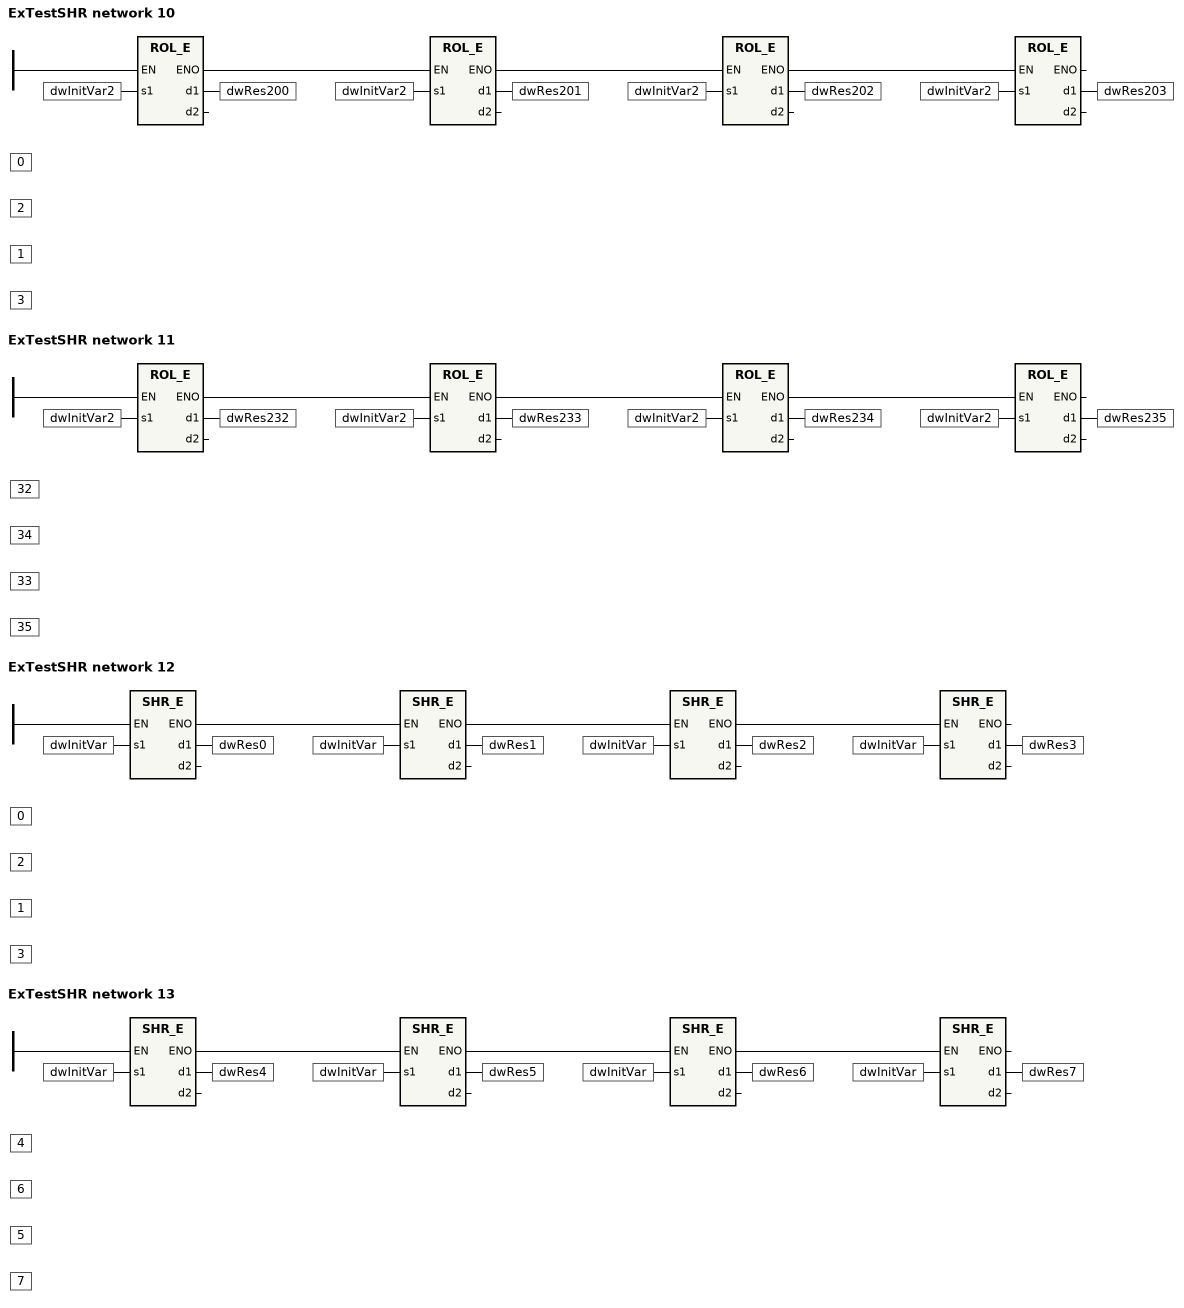
(* network 10 *)
_e1 := ROL_E(TRUE, dwInitVar2, dwRes200, _open);
_e2 := ROL_E(_e1, dwInitVar2, dwRes201, _open);
_e3 := ROL_E(_e2, dwInitVar2, dwRes202, _open);
ROL_E(_e3, dwInitVar2, dwRes203, _open);
(* not connected to any output: 0, 2, 1, 3 *)
(* network 11 *)
_e1 := ROL_E(TRUE, dwInitVar2, dwRes232, _open);
_e2 := ROL_E(_e1, dwInitVar2, dwRes233, _open);
_e3 := ROL_E(_e2, dwInitVar2, dwRes234, _open);
ROL_E(_e3, dwInitVar2, dwRes235, _open);
(* not connected to any output: 32, 34, 33, 35 *)
(* network 12 *)
_e1 := SHR_E(TRUE, dwInitVar, dwRes0, _open);
_e2 := SHR_E(_e1, dwInitVar, dwRes1, _open);
_e3 := SHR_E(_e2, dwInitVar, dwRes2, _open);
SHR_E(_e3, dwInitVar, dwRes3, _open);
(* not connected to any output: 0, 2, 1, 3 *)
(* network 13 *)
_e1 := SHR_E(TRUE, dwInitVar, dwRes4, _open);
_e2 := SHR_E(_e1, dwInitVar, dwRes5, _open);
_e3 := SHR_E(_e2, dwInitVar, dwRes6, _open);
SHR_E(_e3, dwInitVar, dwRes7, _open);
(* not connected to any output: 4, 6, 5, 7 *)
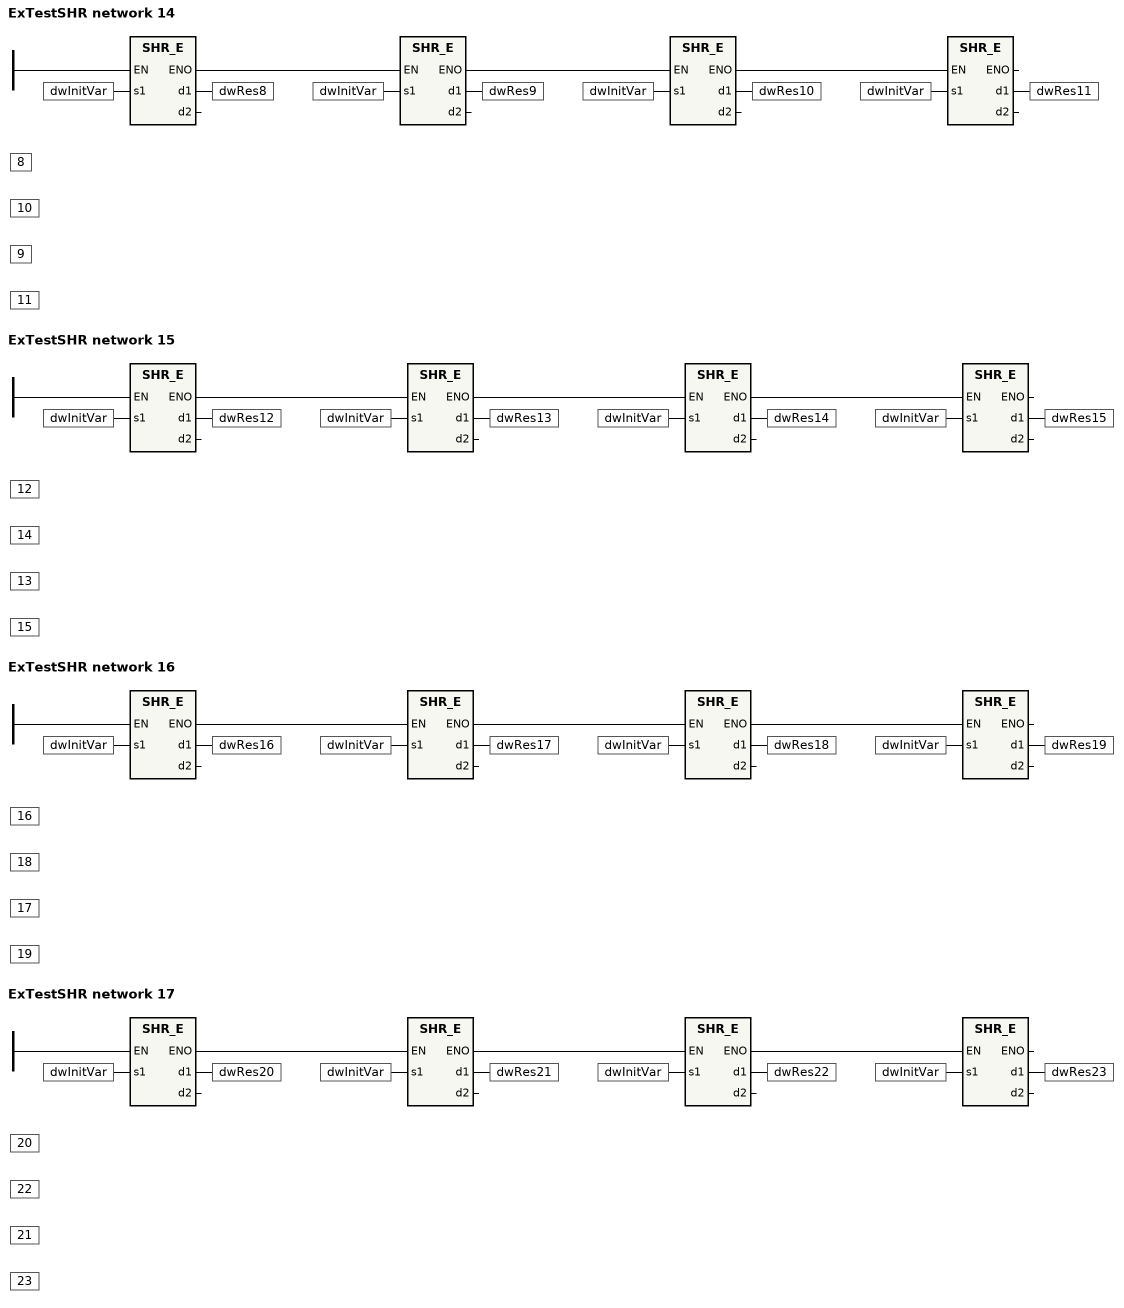
(* network 14 *)
_e1 := SHR_E(TRUE, dwInitVar, dwRes8, _open);
_e2 := SHR_E(_e1, dwInitVar, dwRes9, _open);
_e3 := SHR_E(_e2, dwInitVar, dwRes10, _open);
SHR_E(_e3, dwInitVar, dwRes11, _open);
(* not connected to any output: 8, 10, 9, 11 *)
(* network 15 *)
_e1 := SHR_E(TRUE, dwInitVar, dwRes12, _open);
_e2 := SHR_E(_e1, dwInitVar, dwRes13, _open);
_e3 := SHR_E(_e2, dwInitVar, dwRes14, _open);
SHR_E(_e3, dwInitVar, dwRes15, _open);
(* not connected to any output: 12, 14, 13, 15 *)
(* network 16 *)
_e1 := SHR_E(TRUE, dwInitVar, dwRes16, _open);
_e2 := SHR_E(_e1, dwInitVar, dwRes17, _open);
_e3 := SHR_E(_e2, dwInitVar, dwRes18, _open);
SHR_E(_e3, dwInitVar, dwRes19, _open);
(* not connected to any output: 16, 18, 17, 19 *)
(* network 17 *)
_e1 := SHR_E(TRUE, dwInitVar, dwRes20, _open);
_e2 := SHR_E(_e1, dwInitVar, dwRes21, _open);
_e3 := SHR_E(_e2, dwInitVar, dwRes22, _open);
SHR_E(_e3, dwInitVar, dwRes23, _open);
(* not connected to any output: 20, 22, 21, 23 *)
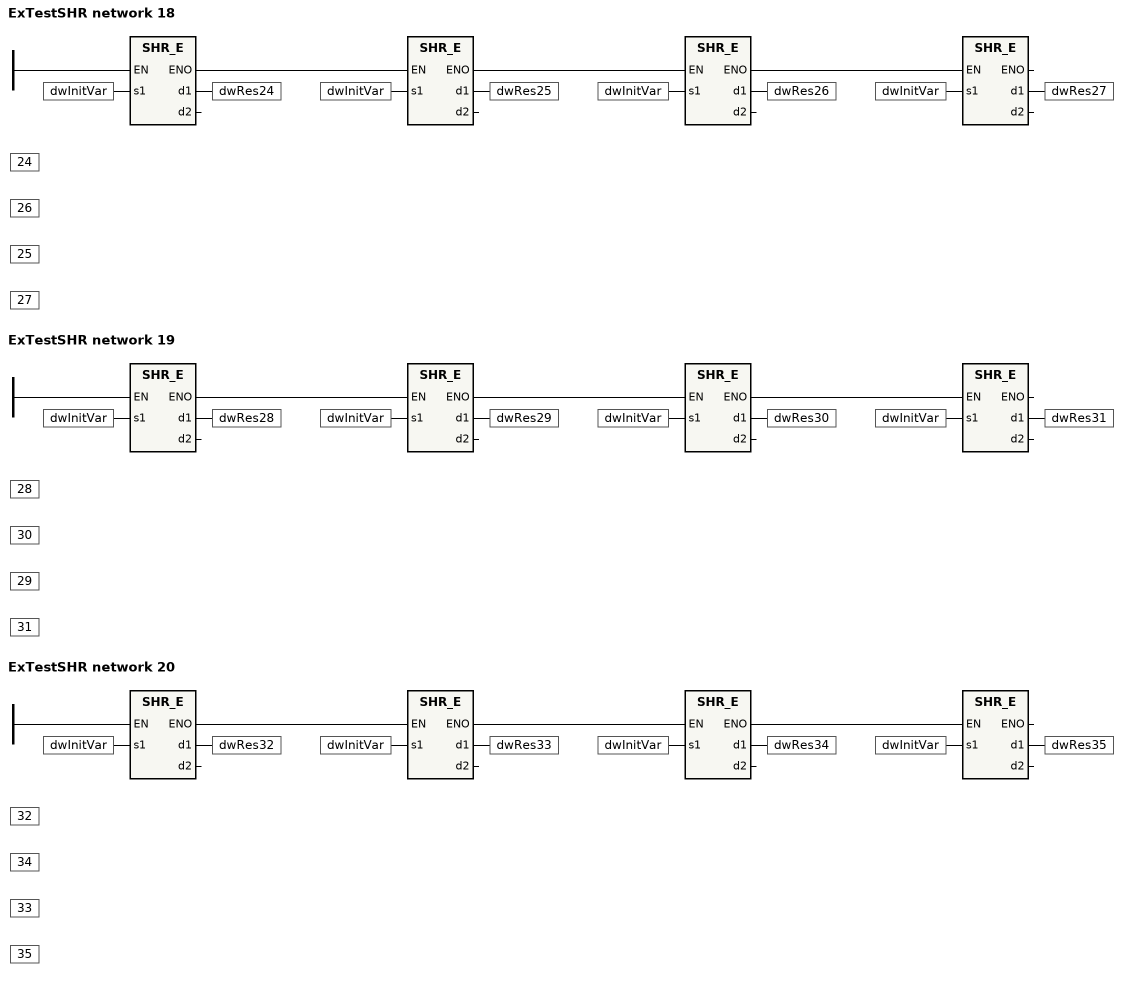
(* network 18 *)
_e1 := SHR_E(TRUE, dwInitVar, dwRes24, _open);
_e2 := SHR_E(_e1, dwInitVar, dwRes25, _open);
_e3 := SHR_E(_e2, dwInitVar, dwRes26, _open);
SHR_E(_e3, dwInitVar, dwRes27, _open);
(* not connected to any output: 24, 26, 25, 27 *)
(* network 19 *)
_e1 := SHR_E(TRUE, dwInitVar, dwRes28, _open);
_e2 := SHR_E(_e1, dwInitVar, dwRes29, _open);
_e3 := SHR_E(_e2, dwInitVar, dwRes30, _open);
SHR_E(_e3, dwInitVar, dwRes31, _open);
(* not connected to any output: 28, 30, 29, 31 *)
(* network 20 *)
_e1 := SHR_E(TRUE, dwInitVar, dwRes32, _open);
_e2 := SHR_E(_e1, dwInitVar, dwRes33, _open);
_e3 := SHR_E(_e2, dwInitVar, dwRes34, _open);
SHR_E(_e3, dwInitVar, dwRes35, _open);
(* not connected to any output: 32, 34, 33, 35 *)
END_PROGRAM

PROGRAM ExError
VAR
  dwInitVar : DWORD;
  dwRes0 : DWORD;
  dwRes1 : DWORD;
  dwRes2 : DWORD;
  dwRes3 : DWORD;
  dwRes4 : DWORD;
  dwRes5 : DWORD;
  dwRes6 : DWORD;
  dwRes7 : DWORD;
  dwRes8 : DWORD;
  dwRes9 : DWORD;
  dwRes10 : DWORD;
  dwRes11 : DWORD;
  dwRes12 : DWORD;
  dwRes13 : DWORD;
  dwRes14 : DWORD;
  dwRes15 : DWORD;
  dwRes16 : DWORD;
  dwRes17 : DWORD;
  dwRes18 : DWORD;
  dwRes19 : DWORD;
  dwRes20 : DWORD;
  dwRes21 : DWORD;
  dwRes22 : DWORD;
  dwRes23 : DWORD;
  dwRes24 : DWORD;
  dwRes25 : DWORD;
  dwRes26 : DWORD;
  dwRes27 : DWORD;
  dwRes28 : DWORD;
  dwRes29 : DWORD;
  dwRes30 : DWORD;
  dwRes31 : DWORD;
  wInitVar : WORD;
  wRes0 : WORD;
  wRes1 : WORD;
  wRes2 : WORD;
  wRes3 : WORD;
  wRes4 : WORD;
  wRes5 : WORD;
  wRes6 : WORD;
  wRes7 : WORD;
  wRes8 : WORD;
  wRes9 : WORD;
  wRes10 : WORD;
  wRes11 : WORD;
  wRes12 : WORD;
  wRes13 : WORD;
  wRes14 : WORD;
  wRes15 : WORD;
  wRes16 : WORD;
  dwRes32 : DWORD;
  dwRes33 : DWORD;
  dwRes34 : DWORD;
  wRes17 : WORD;
  wRes18 : WORD;
  wRes19 : WORD;
  wRes20 : WORD;
  dwRes35 : DWORD;
  dwRes36 : DWORD;
  dwRes100 : DWORD;
  dwRes101 : DWORD;
  dwRes102 : DWORD;
  dwRes103 : DWORD;
  dwRes132 : DWORD;
  dwRes133 : DWORD;
  dwRes134 : DWORD;
  dwRes135 : DWORD;
  dwRes200 : DWORD;
  dwRes201 : DWORD;
  dwRes202 : DWORD;
  dwRes203 : DWORD;
  dwRes232 : DWORD;
  dwRes233 : DWORD;
  dwRes234 : DWORD;
  dwRes235 : DWORD;
  dwInitVar2 : DWORD;
  wInitVar2 : WORD;
END_VAR
(* structured ladder/FBD written out as ST: instructions are called as NAME(EN, inputs, outputs); _pN, _eN, _tN stand for wires *)
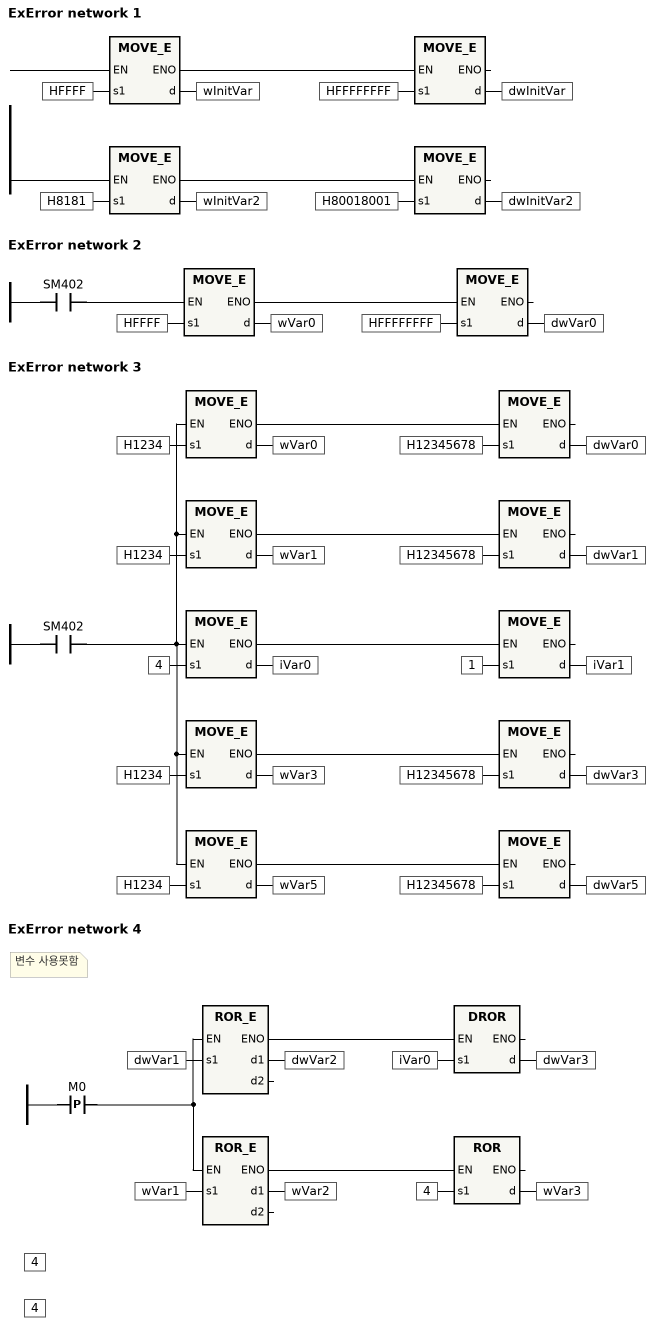
(* network 1 *)
_e1 := MOVE_E(TRUE, HFFFF, wInitVar);
MOVE_E(_e1, HFFFFFFFF, dwInitVar);
_e2 := MOVE_E(TRUE, H8181, wInitVar2);
MOVE_E(_e2, H80018001, dwInitVar2);
(* network 2 *)
_e1 := MOVE_E(SM402, HFFFF, wVar0);
MOVE_E(_e1, HFFFFFFFF, dwVar0);
(* network 3 *)
_e1 := MOVE_E(SM402, H1234, wVar0);
MOVE_E(_e1, H12345678, dwVar0);
_e2 := MOVE_E(SM402, H1234, wVar1);
MOVE_E(_e2, H12345678, dwVar1);
_e3 := MOVE_E(SM402, 4, iVar0);
MOVE_E(_e3, 1, iVar1);
_e4 := MOVE_E(SM402, H1234, wVar3);
MOVE_E(_e4, H12345678, dwVar3);
_e5 := MOVE_E(SM402, H1234, wVar5);
MOVE_E(_e5, H12345678, dwVar5);
(* network 4 *)
(* 변수 사용못함 *)
_p1 := LDP(TRUE, M0);
_e2 := ROR_E(_p1, dwVar1, dwVar2, _open);
DROR(_e2, iVar0, dwVar3);
_e3 := ROR_E(_p1, wVar1, wVar2, _open);
ROR(_e3, 4, wVar3);
(* not connected to any output: 4, 4 *)
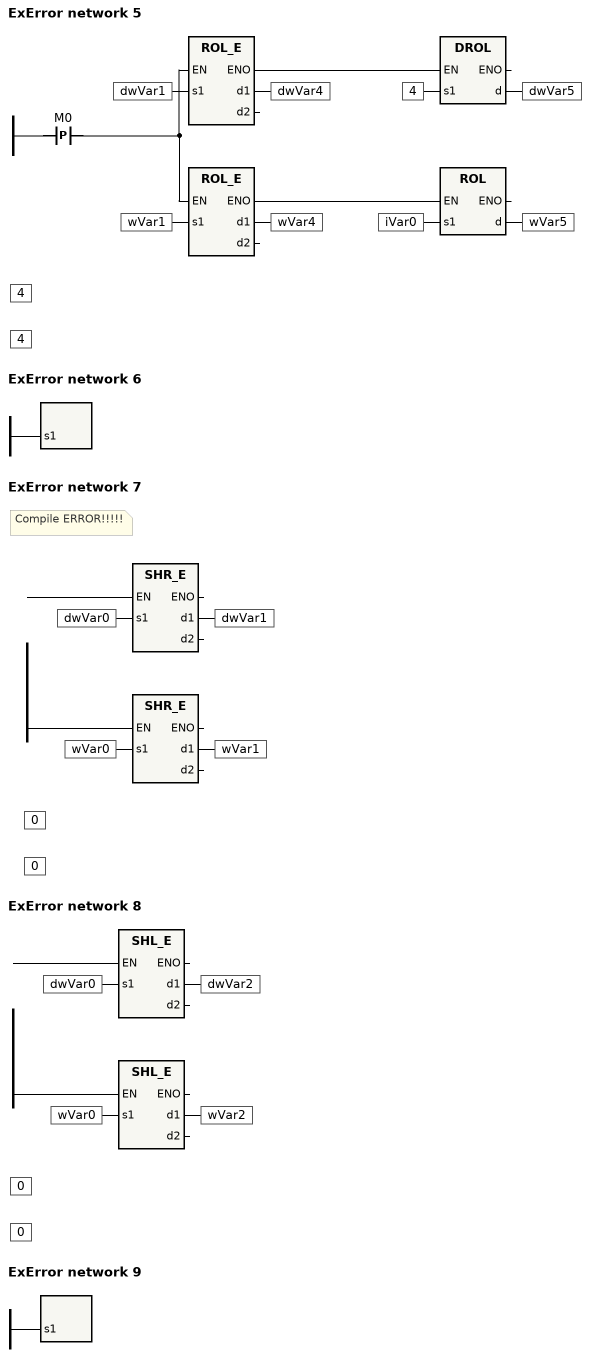
(* network 5 *)
_p1 := LDP(TRUE, M0);
_e2 := ROL_E(_p1, dwVar1, dwVar4, _open);
DROL(_e2, 4, dwVar5);
_e3 := ROL_E(_p1, wVar1, wVar4, _open);
ROL(_e3, iVar0, wVar5);
(* not connected to any output: 4, 4 *)
(* network 6 *)
(* element kind 10  <- TRUE *)
(* network 7 *)
(* Compile ERROR!!!!! *)
SHR_E(TRUE, dwVar0, dwVar1, _open);
SHR_E(TRUE, wVar0, wVar1, _open);
(* not connected to any output: 0, 0 *)
(* network 8 *)
SHL_E(TRUE, dwVar0, dwVar2, _open);
SHL_E(TRUE, wVar0, wVar2, _open);
(* not connected to any output: 0, 0 *)
(* network 9 *)
(* element kind 10  <- TRUE *)
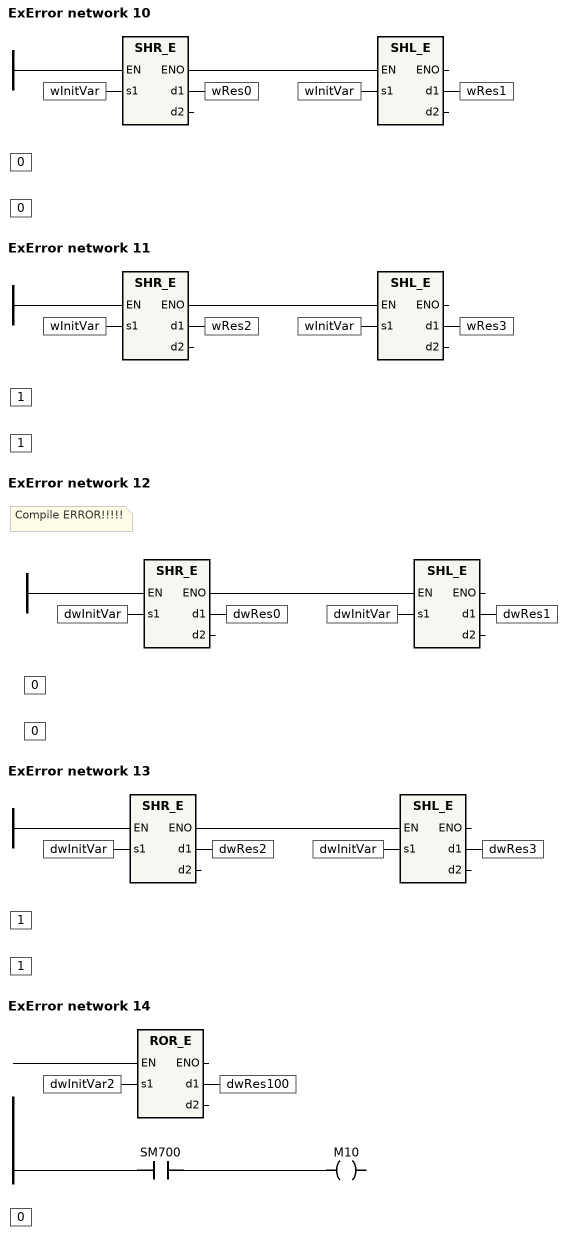
(* network 10 *)
_e1 := SHR_E(TRUE, wInitVar, wRes0, _open);
SHL_E(_e1, wInitVar, wRes1, _open);
(* not connected to any output: 0, 0 *)
(* network 11 *)
_e1 := SHR_E(TRUE, wInitVar, wRes2, _open);
SHL_E(_e1, wInitVar, wRes3, _open);
(* not connected to any output: 1, 1 *)
(* network 12 *)
(* Compile ERROR!!!!! *)
_e1 := SHR_E(TRUE, dwInitVar, dwRes0, _open);
SHL_E(_e1, dwInitVar, dwRes1, _open);
(* not connected to any output: 0, 0 *)
(* network 13 *)
_e1 := SHR_E(TRUE, dwInitVar, dwRes2, _open);
SHL_E(_e1, dwInitVar, dwRes3, _open);
(* not connected to any output: 1, 1 *)
(* network 14 *)
ROR_E(TRUE, dwInitVar2, dwRes100, _open);
M10 := SM700;
(* not connected to any output: 0 *)
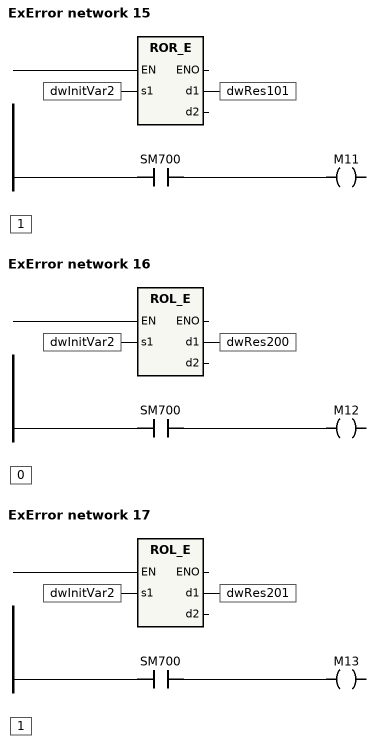
(* network 15 *)
ROR_E(TRUE, dwInitVar2, dwRes101, _open);
M11 := SM700;
(* not connected to any output: 1 *)
(* network 16 *)
ROL_E(TRUE, dwInitVar2, dwRes200, _open);
M12 := SM700;
(* not connected to any output: 0 *)
(* network 17 *)
ROL_E(TRUE, dwInitVar2, dwRes201, _open);
M13 := SM700;
(* not connected to any output: 1 *)
END_PROGRAM
